SUBAPPLICATION ein (* Subapplication Type *)
  (* Standard: 61499-2 *)
  (* Version 1.0, 2023-02-07, franz *)
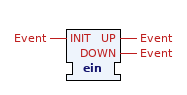
  EVENT_INPUT
    INIT;
  END_EVENT
  EVENT_OUTPUT
    UP;
    DOWN;
  END_EVENT
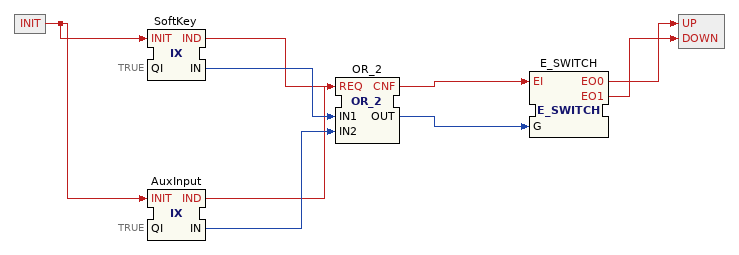
  FBS
    SoftKey : IX(QI := TRUE);
    AuxInput : IX(QI := TRUE);
    OR_2 : OR_2;
    E_SWITCH : E_SWITCH;
  END_FBS
  EVENT_CONNECTIONS
    INIT TO SoftKey.INIT;
    INIT TO AuxInput.INIT;
    SoftKey.IND TO OR_2.REQ;
    AuxInput.IND TO OR_2.REQ;
    OR_2.CNF TO E_SWITCH.EI;
    E_SWITCH.EO0 TO UP;
    E_SWITCH.EO1 TO DOWN;
  END_CONNECTIONS
  DATA_CONNECTIONS
    SoftKey.IN TO OR_2.IN1;
    AuxInput.IN TO OR_2.IN2;
    OR_2.OUT TO E_SWITCH.G;
  END_CONNECTIONS
END_SUBAPPLICATION
